ABB RAPID module: 002C9C5E

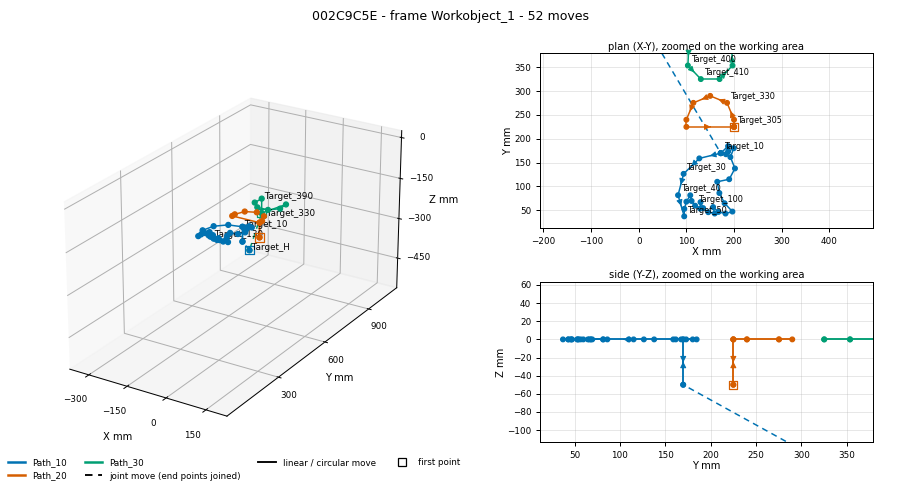
[picture p0: tool path of 002C9C5E in frame Workobject_1, 52 of 52 moves have a stored position in this frame; points joined in program order, loops and branches not executed]
MODULE Module1
        CONST robtarget Target_H:=[[-350,1055.651275023,-538.588646413],[0.701057385,-0.092295956,-0.092295956,-0.701057385],[0,0,0,0],[9E+09,9E+09,9E+09,9E+09,9E+09,9E+09]];
    CONST robtarget Target_10:=[[172.145654378,169.721037846,0],[0.015654757,0,0,0.999877457],[1,-2,1,0],[9E+09,9E+09,9E+09,9E+09,9E+09,9E+09]];
    CONST robtarget Target_20:=[[127.176015411,158.806349071,0],[0.015654757,0,0,0.999877457],[1,-2,1,0],[9E+09,9E+09,9E+09,9E+09,9E+09,9E+09]];
    CONST robtarget Target_30:=[[94.179068929,126.362545613,0],[0.015654757,0,0,0.999877457],[1,-2,1,0],[9E+09,9E+09,9E+09,9E+09,9E+09,9E+09]];
    CONST robtarget Target_40:=[[82.505775243,81.583833322,0],[0.015654757,0,0,0.999877457],[1,-2,1,0],[9E+09,9E+09,9E+09,9E+09,9E+09,9E+09]];
    CONST robtarget Target_50:=[[95.464213358,37.159991282,0],[0.015654757,0,0,0.999877457],[1,-2,1,0],[9E+09,9E+09,9E+09,9E+09,9E+09,9E+09]];
    CONST robtarget Target_60:=[[95.659015698,52.859355196,0],[0.015654757,0,0,0.999877457],[1,-2,1,0],[9E+09,9E+09,9E+09,9E+09,9E+09,9E+09]];
    CONST robtarget Target_70:=[[99.986563128,67.9517476,0],[0.015654757,0,0,0.999877457],[1,-2,1,0],[9E+09,9E+09,9E+09,9E+09,9E+09,9E+09]];
    CONST robtarget Target_80:=[[108.140548997,81.368919049,0],[0.015654757,0,0,0.999877457],[1,-2,1,0],[9E+09,9E+09,9E+09,9E+09,9E+09,9E+09]];
    CONST robtarget Target_90:=[[110.943419364,69.425655071,0],[0.015654757,0,0,0.999877457],[1,-2,1,0],[9E+09,9E+09,9E+09,9E+09,9E+09,9E+09]];
    CONST robtarget Target_100:=[[118.270530204,59.586392727,0],[0.015654757,0,0,0.999877457],[1,-2,1,0],[9E+09,9E+09,9E+09,9E+09,9E+09,9E+09]];
    CONST robtarget Target_110:=[[128.909818396,53.478759508,0],[0.015654757,0,0,0.999877457],[1,-2,1,0],[9E+09,9E+09,9E+09,9E+09,9E+09,9E+09]];
    CONST robtarget Target_120:=[[129.685602376,67.032677318,0],[0.015654757,0,0,0.999877457],[1,-2,1,0],[9E+09,9E+09,9E+09,9E+09,9E+09,9E+09]];
    CONST robtarget Target_130:=[[135.242270658,54.463630271,0],[0.015654757,0,0,0.999877457],[1,-2,1,0],[9E+09,9E+09,9E+09,9E+09,9E+09,9E+09]];
    CONST robtarget Target_140:=[[145.944316156,45.842509218,0],[0.015654757,0,0,0.999877457],[1,-2,1,0],[9E+09,9E+09,9E+09,9E+09,9E+09,9E+09]];
    CONST robtarget Target_150:=[[159.408253951,43.089350102,0],[0.015654757,0,0,0.999877457],[1,-2,1,0],[9E+09,9E+09,9E+09,9E+09,9E+09,9E+09]];
    CONST robtarget Target_160:=[[156.13873613,56.659281011,0],[0.015654757,0,0,0.999877457],[1,-2,1,0],[9E+09,9E+09,9E+09,9E+09,9E+09,9E+09]];
    CONST robtarget Target_170:=[[167.339659667,46.46756084,0],[0.015654757,0,0,0.999877457],[1,-2,1,0],[9E+09,9E+09,9E+09,9E+09,9E+09,9E+09]];
    CONST robtarget Target_180:=[[182.086391819,43.022892643,0],[0.015654757,0,0,0.999877457],[1,-1,1,0],[9E+09,9E+09,9E+09,9E+09,9E+09,9E+09]];
    CONST robtarget Target_190:=[[196.643218036,47.197896671,0],[0.015654757,0,0,0.999877457],[1,-1,1,0],[9E+09,9E+09,9E+09,9E+09,9E+09,9E+09]];
    CONST robtarget Target_200:=[[180.134939682,64.681155269,0],[0.015654757,0,0,0.999877457],[1,-2,1,0],[9E+09,9E+09,9E+09,9E+09,9E+09,9E+09]];
    CONST robtarget Target_210:=[[169.208263421,86.100663464,0],[0.015654757,0,0,0.999877457],[1,-2,1,0],[9E+09,9E+09,9E+09,9E+09,9E+09,9E+09]];
    CONST robtarget Target_220:=[[164.744756678,109.728289095,0],[0.015654757,0,0,0.999877457],[1,-2,1,0],[9E+09,9E+09,9E+09,9E+09,9E+09,9E+09]];
    CONST robtarget Target_230:=[[189.86479429,115.046784411,0],[0.015654757,0,0,0.999877457],[1,-2,1,0],[9E+09,9E+09,9E+09,9E+09,9E+09,9E+09]];
    CONST robtarget Target_240:=[[201.945805105,137.70405388,0],[0.015654757,0,0,0.999877457],[1,-2,1,0],[9E+09,9E+09,9E+09,9E+09,9E+09,9E+09]];
    CONST robtarget Target_250:=[[192.36364797,161.525996428,0],[0.015654757,0,0,0.999877457],[1,-2,1,0],[9E+09,9E+09,9E+09,9E+09,9E+09,9E+09]];
    CONST robtarget Target_260:=[[199.538662434,180.200691671,0],[0.015654757,0,0,0.999877457],[1,-2,1,0],[9E+09,9E+09,9E+09,9E+09,9E+09,9E+09]];
    CONST robtarget Target_270:=[[187.501772235,172.981329375,0],[0.015654757,0,0,0.999877457],[1,-2,1,0],[9E+09,9E+09,9E+09,9E+09,9E+09,9E+09]];
    CONST robtarget Target_280:=[[183.067776679,167.478919652,0],[0.015654757,0,0,0.999877457],[1,-2,1,0],[9E+09,9E+09,9E+09,9E+09,9E+09,9E+09]];
    CONST robtarget Target_290:=[[187.548582623,184.533188144,0],[0.015654757,0,0,0.999877457],[1,-2,1,0],[9E+09,9E+09,9E+09,9E+09,9E+09,9E+09]];
    CONST robtarget Target_300:=[[172.145654378,169.721037846,0],[0.015654757,0,0,0.999877457],[1,-2,1,0],[9E+09,9E+09,9E+09,9E+09,9E+09,9E+09]];
    CONST robtarget Target_305:=[[200,225,-50],[0.015654757,0,0,0.999877457],[1,-2,1,0],[9E+09,9E+09,9E+09,9E+09,9E+09,9E+09]];
    CONST robtarget Target_310:=[[200,225,0],[0.015654757,0,0,0.999877457],[1,-2,1,0],[9E+09,9E+09,9E+09,9E+09,9E+09,9E+09]];
    CONST robtarget Target_320:=[[200,240,0],[0.015654757,0,0,0.999877457],[1,-2,1,0],[9E+09,9E+09,9E+09,9E+09,9E+09,9E+09]];
    CONST robtarget Target_330:=[[185.355339059,275.355339059,0],[0.015654757,0,0,0.999877457],[1,-2,1,0],[9E+09,9E+09,9E+09,9E+09,9E+09,9E+09]];
    CONST robtarget Target_340:=[[150,290,0],[0.015654757,0,0,0.999877457],[1,-2,1,0],[9E+09,9E+09,9E+09,9E+09,9E+09,9E+09]];
    CONST robtarget Target_350:=[[114.644660941,275.355339059,0],[0.015654757,0,0,0.999877457],[1,-2,1,0],[9E+09,9E+09,9E+09,9E+09,9E+09,9E+09]];
    CONST robtarget Target_360:=[[100,240,0],[0.015654757,0,0,0.999877457],[1,-2,1,0],[9E+09,9E+09,9E+09,9E+09,9E+09,9E+09]];
    CONST robtarget Target_370:=[[100,225,0],[0.015654757,0,0,0.999877457],[1,-2,1,0],[9E+09,9E+09,9E+09,9E+09,9E+09,9E+09]];
    CONST robtarget Target_380:=[[200,225,0],[0.015654757,0,0,0.999877457],[1,-2,1,0],[9E+09,9E+09,9E+09,9E+09,9E+09,9E+09]];
    CONST robtarget Target_385:=[[105,392.991805459,-50],[0.015654757,0,0,0.999877457],[1,-2,1,0],[9E+09,9E+09,9E+09,9E+09,9E+09,9E+09]];
    CONST robtarget Target_390:=[[105,392.991805459,0],[0.015654757,0,0,0.999877457],[1,-2,1,0],[9E+09,9E+09,9E+09,9E+09,9E+09,9E+09]];
    CONST robtarget Target_400:=[[103.164813866,353.691159257,0],[0.015654757,0,0,0.999877457],[1,-2,1,0],[9E+09,9E+09,9E+09,9E+09,9E+09,9E+09]];
    CONST robtarget Target_410:=[[130.328264565,325.22968273,0],[0.015654757,0,0,0.999877457],[1,-2,1,0],[9E+09,9E+09,9E+09,9E+09,9E+09,9E+09]];
    CONST robtarget Target_420:=[[169.671735435,325.22968273,0],[0.015654757,0,0,0.999877457],[1,-2,1,0],[9E+09,9E+09,9E+09,9E+09,9E+09,9E+09]];
    CONST robtarget Target_430:=[[196.835186134,353.691159257,0],[0.015654757,0,0,0.999877457],[1,-2,1,0],[9E+09,9E+09,9E+09,9E+09,9E+09,9E+09]];
    CONST robtarget Target_440:=[[195,392.991805459,0],[0.015654757,0,0,0.999877457],[1,-2,1,0],[9E+09,9E+09,9E+09,9E+09,9E+09,9E+09]];
!***********************************************************
    !
    ! M?dulo:  Module1
    !
    ! Descripción:
    !   <Introduzca la descripción aquí>
    !
    ! Autor: ASUS
    !
    ! Versión: 1.0
    !
    !***********************************************************


    !***********************************************************
    !
    ! Procedimiento Main
    !
    !   Este es el punto de entrada de su programa
    !
    !***********************************************************
    PROC main()
        !Add your code here
        first;
    ENDPROC
    PROC Path_10()
        MoveJ Target_H,v600,z5,THerramienta\WObj:=Workobject_1;
        MoveJ [[172.145654378,169.721037846,-50],[0.015654757,0,0,0.999877457],[1,-2,1,0],[9E+09,9E+09,9E+09,9E+09,9E+09,9E+09]],v400,z5,THerramienta\WObj:=Workobject_1;
        MoveL Target_10,v200,z0,THerramienta\WObj:=Workobject_1;
        MoveL Target_20,v200,z5,THerramienta\WObj:=Workobject_1;
        MoveL Target_30,v200,z5,THerramienta\WObj:=Workobject_1;
        MoveL Target_40,v200,z5,THerramienta\WObj:=Workobject_1;
        MoveL Target_50,v200,z5,THerramienta\WObj:=Workobject_1;
        MoveL Target_60,v200,z5,THerramienta\WObj:=Workobject_1;
        MoveL Target_70,v200,z5,THerramienta\WObj:=Workobject_1;
        MoveL Target_80,v200,z5,THerramienta\WObj:=Workobject_1;
        MoveL Target_90,v200,z5,THerramienta\WObj:=Workobject_1;
        MoveL Target_100,v200,z5,THerramienta\WObj:=Workobject_1;
        MoveL Target_110,v200,z5,THerramienta\WObj:=Workobject_1;
        MoveL Target_120,v200,z5,THerramienta\WObj:=Workobject_1;
        MoveL Target_130,v200,z5,THerramienta\WObj:=Workobject_1;
        MoveL Target_140,v200,z5,THerramienta\WObj:=Workobject_1;
        MoveL Target_150,v200,z5,THerramienta\WObj:=Workobject_1;
        MoveL Target_160,v200,z5,THerramienta\WObj:=Workobject_1;
        MoveL Target_170,v200,z5,THerramienta\WObj:=Workobject_1;
        MoveL Target_180,v200,z5,THerramienta\WObj:=Workobject_1;
        MoveL Target_190,v200,z5,THerramienta\WObj:=Workobject_1;
        MoveL Target_200,v200,z5,THerramienta\WObj:=Workobject_1;
        MoveL Target_210,v200,z5,THerramienta\WObj:=Workobject_1;
        MoveL Target_220,v200,z5,THerramienta\WObj:=Workobject_1;
        MoveL Target_230,v200,z5,THerramienta\WObj:=Workobject_1;
        MoveL Target_240,v200,z5,THerramienta\WObj:=Workobject_1;
        MoveL Target_250,v200,z5,THerramienta\WObj:=Workobject_1;
        MoveL Target_260,v200,z5,THerramienta\WObj:=Workobject_1;
        MoveL Target_270,v200,z5,THerramienta\WObj:=Workobject_1;
        MoveL Target_280,v200,z5,THerramienta\WObj:=Workobject_1;
        MoveL Target_290,v200,z5,THerramienta\WObj:=Workobject_1;
        MoveL Target_300,v200,z0,THerramienta\WObj:=Workobject_1;
        MoveL [[172.145654378,169.721037846,-50],[0.015654757,0,0,0.999877457],[1,-2,1,0],[9E+09,9E+09,9E+09,9E+09,9E+09,9E+09]],v200,z100,THerramienta\WObj:=Workobject_1;
    ENDPROC
    PROC Path_20()
        MoveJ Target_305,v400,z5,THerramienta\WObj:=Workobject_1;
        MoveL Target_310,v200,z0,THerramienta\WObj:=Workobject_1;
        MoveL Target_320,v200,z5,THerramienta\WObj:=Workobject_1;
        MoveL Target_330,v200,z5,THerramienta\WObj:=Workobject_1;
        MoveL Target_340,v200,z5,THerramienta\WObj:=Workobject_1;
        MoveL Target_350,v200,z5,THerramienta\WObj:=Workobject_1;
        MoveL Target_360,v200,z5,THerramienta\WObj:=Workobject_1;
        MoveL Target_370,v200,z5,THerramienta\WObj:=Workobject_1;
        MoveL Target_380,v200,z0,THerramienta\WObj:=Workobject_1;
        MoveL Target_305,v200,z5,THerramienta\WObj:=Workobject_1;
    ENDPROC
    PROC first()
        Path_10;
        Path_20;
        Path_30;
    ENDPROC
    PROC Path_30()
        MoveL Target_385,v200,z5,THerramienta\WObj:=Workobject_1;
        MoveL Target_390,v200,z5,THerramienta\WObj:=Workobject_1;
        MoveL Target_400,v200,z5,THerramienta\WObj:=Workobject_1;
        MoveL Target_410,v200,z5,THerramienta\WObj:=Workobject_1;
        MoveL Target_420,v200,z5,THerramienta\WObj:=Workobject_1;
        MoveL Target_430,v200,z5,THerramienta\WObj:=Workobject_1;
        MoveL Target_440,v200,z5,THerramienta\WObj:=Workobject_1;
        MoveL Target_385,v200,z5,THerramienta\WObj:=Workobject_1;
        MoveJ Target_H,v600,z5,THerramienta\WObj:=Workobject_1;
    ENDPROC
ENDMODULE
